FUNCTION_BLOCK FB_HeatingElement EXTENDS FB_ComponentBase IMPLEMENTS I_HeatingElement
VAR
	_enabled 	: BOOL;				
	_output  	AT %Q* : BOOL;
	_state		: E_State := ABORTED;
END_VAR

///////////////////////////////////////////////////////////////////////////////////////////
//
//	States:
//	Before initializing: ABORTED
//	Once initialized, disabled: STOPPED
//	Once initialized, enabled: IDLE
//	Once enabled, PowerOn: EXECUTE
//	Once enabled, PowerOff: IDLE
//
//
//

METHOD Disable
_enabled := FALSE;
PowerOff();
_State := STOPPED;
END_METHOD

METHOD Enable
_enabled := TRUE;
_State := IDLE;
END_METHOD

METHOD Init
_enabled := FALSE;
PowerOff();
_State := STOPPED;
END_METHOD

PROPERTY isHeating : BOOL
GET
isHeating := _output;
END_GET
END_PROPERTY

METHOD PowerOff : BOOL
_output := FALSE;
_State := IDLE;
END_METHOD

METHOD PowerOn : BOOL
IF _enabled THEN
	_output := TRUE;
	_State := EXECUTE;
END_IF
END_METHOD

PROPERTY State : E_State
GET
END_GET
END_PROPERTY

END_FUNCTION_BLOCK

(* stored: Version 1.1.0.1
   POU FB_HeatingElement: Id {96f3a9f0-42cb-4156-af01-85514b68b235}, SpecialFunc None
   Method Disable: Id {27106d6a-4292-4cc8-942c-49ea21dc9af7}
   Method Enable: Id {47265e9f-e11f-4c11-b54d-8bcef40f5661}
   Method Init: Id {ded90bbb-33b1-446f-bf83-145ce1aa46d0}
   Property isHeating: Id {6d5582a3-e5bc-4b51-bb49-67faeb1b2e52}
   Get Get: Id {1736e8f1-3528-439d-9478-9015bf72eac0}
   Method PowerOff: Id {59908f49-21fe-4588-a981-65362939a12a}
   Method PowerOn: Id {c293af04-ea37-4eab-a009-fd29fc83aa9e}
   Property State: Id {2e7b7cfe-045f-4df6-a825-628e66d97828}
   Get Get: Id {9cc6bab6-0bab-454c-b569-d6ca41ccd59e} *)
